Universal Robots PolyScope program: Ruch4MS.urp

Program Ruch4MS (installation=default directory=/programs/usbdisk createdIn=3.15.8.106339 lastSavedIn=3.15.8.106339 robotSerialNumber=2020330428)
Calibrated DH parameters: a=[0.000029, -0.241913, -0.128453, -0.000049, -0.000012, 0]; d=[0.151842, -4.082088, 33.504745, -29.309875, 0.08529, 0.082285]; alpha=[1.571059, -0.006644, 0.005794, 1.571984, -1.571997, 0]; deltaTheta=[-0.000032, 0.111537, 0.813391, -0.924919, 0.000036, 0.000016]
Robot Program (runOnlyOnce=false)
  MoveJ speed 60 deg/s, acceleration 120 deg/s^2 (useActiveTCP=true)
    Waypoint Punkt_orienta_1: TCP in base x=-156.761 y=-113.895 z=693.367 mm, rx=-1.2064 ry=-1.2136 rz=1.2088 rad; joints [-0.002, -90.003, -0.003, -90, -90, 0.003] deg; flange x=-81.761 y=-113.664 z=693.448 mm, rx=-1.2064 ry=-1.2136 rz=1.2088 rad
    Waypoint Punkt_orienta_2: TCP in base x=157.696 y=-112.222 z=523.13 mm, rx=1.211 ry=1.2081 rz=1.216 rad; joints [0.001, -90.004, -0.003, -270, -90, 0.004] deg; flange x=82.696 y=-112.451 z=523.049 mm, rx=1.211 ry=1.2081 rz=1.216 rad
